{attribute addProperty BoxType "EL3423-0000-0017"}
{attribute addProperty Id "Reset_IntervalAT %Q*BOOL81"}
{attribute addProperty CRC "2882377394"}
{attribute addProperty SizeInBites "8"}
{attribute addProperty SizeInBytes "1"}
TYPE Total_Interval_ABCD96B2 :
STRUCT
	{attribute addProperty Name "Reset_Interval"}
	Reset_Interval AT %Q* : BOOL;
END_STRUCT
END_TYPE

(* stored: Version 1.2.0.0, ProductVersion 3.1.4024.9
   DUT Total_Interval_ABCD96B2: Id {7479eaf5-f258-45e0-a39a-7dfdae16f487} *)
